PROGRAM MAIN
VAR
END_VAR

END_PROGRAM

(* stored: Version 1.1.0.1
   POU MAIN: Id {3b393217-f6cc-4465-870d-8b543b9de436} *)
